(* PLC project PinDiagnosis, Hydac System GmbH PdtCodeBuilder.dll 1.2.7.80 *)
(* stored: companyURL http://www.hydac.com/, contentDescription This content was automatically generated. Please do not edit., creationDateTime 2025-04-18T16:40:50.760, version 1.0.0 *)

VAR_GLOBAL CONSTANT  (* Pins *)
  gc_PinList_C0 : ARRAY[0..95] OF POINTER TO TControllerPinProperties := [ADR(gc_Pin_C0_1), ADR(gc_Pin_C0_2), ADR(gc_Pin_C0_3), ADR(gc_Pin_C0_4), ADR(gc_Pin_C0_5), ADR(gc_Pin_C0_6), ADR(gc_Pin_C0_7), ADR(gc_Pin_C0_8), ADR(gc_Pin_C0_9), ADR(gc_Pin_C0_10), ADR(gc_Pin_C0_11), ADR(gc_Pin_C0_12), ADR(gc_Pin_C0_13), ADR(gc_Pin_C0_14), ADR(gc_Pin_C0_15), ADR(gc_Pin_C0_16), ADR(gc_Pin_C0_17), ADR(gc_Pin_C0_18), ADR(gc_Pin_C0_19), ADR(gc_Pin_C0_20), ADR(gc_Pin_C0_21), ADR(gc_Pin_C0_22), ADR(gc_Pin_C0_23), ADR(gc_Pin_C0_24), ADR(gc_Pin_C0_25), ADR(gc_Pin_C0_26), ADR(gc_Pin_C0_27), ADR(gc_Pin_C0_28), ADR(gc_Pin_C0_29), ADR(gc_Pin_C0_30), ADR(gc_Pin_C0_31), ADR(gc_Pin_C0_32), ADR(gc_Pin_C0_33), ADR(gc_Pin_C0_34), ADR(gc_Pin_C0_35), ADR(gc_Pin_C0_36), ADR(gc_Pin_C0_37), ADR(gc_Pin_C0_38), ADR(gc_Pin_C0_39), ADR(gc_Pin_C0_40), ADR(gc_Pin_C0_41), ADR(gc_Pin_C0_42), ADR(gc_Pin_C0_43), ADR(gc_Pin_C0_44), ADR(gc_Pin_C0_45), ADR(gc_Pin_C0_46), ADR(gc_Pin_C0_47), ADR(gc_Pin_C0_48), ADR(gc_Pin_C0_49), ADR(gc_Pin_C0_50), ADR(gc_Pin_C0_51), ADR(gc_Pin_C0_52), ADR(gc_Pin_C0_53), ADR(gc_Pin_C0_54), ADR(gc_Pin_C0_55), ADR(gc_Pin_C0_56), ADR(gc_Pin_C0_57), ADR(gc_Pin_C0_58), ADR(gc_Pin_C0_59), ADR(gc_Pin_C0_60), ADR(gc_Pin_C0_61), ADR(gc_Pin_C0_62), ADR(gc_Pin_C0_63), ADR(gc_Pin_C0_64), ADR(gc_Pin_C0_65), ADR(gc_Pin_C0_66), ADR(gc_Pin_C0_67), ADR(gc_Pin_C0_68), ADR(gc_Pin_C0_69), ADR(gc_Pin_C0_70), ADR(gc_Pin_C0_71), ADR(gc_Pin_C0_72), ADR(gc_Pin_C0_73), ADR(gc_Pin_C0_74), ADR(gc_Pin_C0_75), ADR(gc_Pin_C0_76), ADR(gc_Pin_C0_77), ADR(gc_Pin_C0_78), ADR(gc_Pin_C0_79), ADR(gc_Pin_C0_80), ADR(gc_Pin_C0_81), ADR(gc_Pin_C0_82), ADR(gc_Pin_C0_83), ADR(gc_Pin_C0_84), ADR(gc_Pin_C0_85), ADR(gc_Pin_C0_86), ADR(gc_Pin_C0_87), ADR(gc_Pin_C0_88), ADR(gc_Pin_C0_89), ADR(gc_Pin_C0_90), ADR(gc_Pin_C0_91), ADR(gc_Pin_C0_92), ADR(gc_Pin_C0_93), ADR(gc_Pin_C0_94), ADR(gc_Pin_C0_95), ADR(gc_Pin_C0_96)];
  gc_ControllerPinConfig_C0 : TControllerPinConfig := (EcuSA := 16#20, EcuName := 'C0', PinCount := 96, Pins := ADR(gc_PinList_C0));
  gc_PinList_C1 : ARRAY[0..95] OF POINTER TO TControllerPinProperties := [ADR(gc_Pin_C1_1), ADR(gc_Pin_C1_2), ADR(gc_Pin_C1_3), ADR(gc_Pin_C1_4), ADR(gc_Pin_C1_5), ADR(gc_Pin_C1_6), ADR(gc_Pin_C1_7), ADR(gc_Pin_C1_8), ADR(gc_Pin_C1_9), ADR(gc_Pin_C1_10), ADR(gc_Pin_C1_11), ADR(gc_Pin_C1_12), ADR(gc_Pin_C1_13), ADR(gc_Pin_C1_14), ADR(gc_Pin_C1_15), ADR(gc_Pin_C1_16), ADR(gc_Pin_C1_17), ADR(gc_Pin_C1_18), ADR(gc_Pin_C1_19), ADR(gc_Pin_C1_20), ADR(gc_Pin_C1_21), ADR(gc_Pin_C1_22), ADR(gc_Pin_C1_23), ADR(gc_Pin_C1_24), ADR(gc_Pin_C1_25), ADR(gc_Pin_C1_26), ADR(gc_Pin_C1_27), ADR(gc_Pin_C1_28), ADR(gc_Pin_C1_29), ADR(gc_Pin_C1_30), ADR(gc_Pin_C1_31), ADR(gc_Pin_C1_32), ADR(gc_Pin_C1_33), ADR(gc_Pin_C1_34), ADR(gc_Pin_C1_35), ADR(gc_Pin_C1_36), ADR(gc_Pin_C1_37), ADR(gc_Pin_C1_38), ADR(gc_Pin_C1_39), ADR(gc_Pin_C1_40), ADR(gc_Pin_C1_41), ADR(gc_Pin_C1_42), ADR(gc_Pin_C1_43), ADR(gc_Pin_C1_44), ADR(gc_Pin_C1_45), ADR(gc_Pin_C1_46), ADR(gc_Pin_C1_47), ADR(gc_Pin_C1_48), ADR(gc_Pin_C1_49), ADR(gc_Pin_C1_50), ADR(gc_Pin_C1_51), ADR(gc_Pin_C1_52), ADR(gc_Pin_C1_53), ADR(gc_Pin_C1_54), ADR(gc_Pin_C1_55), ADR(gc_Pin_C1_56), ADR(gc_Pin_C1_57), ADR(gc_Pin_C1_58), ADR(gc_Pin_C1_59), ADR(gc_Pin_C1_60), ADR(gc_Pin_C1_61), ADR(gc_Pin_C1_62), ADR(gc_Pin_C1_63), ADR(gc_Pin_C1_64), ADR(gc_Pin_C1_65), ADR(gc_Pin_C1_66), ADR(gc_Pin_C1_67), ADR(gc_Pin_C1_68), ADR(gc_Pin_C1_69), ADR(gc_Pin_C1_70), ADR(gc_Pin_C1_71), ADR(gc_Pin_C1_72), ADR(gc_Pin_C1_73), ADR(gc_Pin_C1_74), ADR(gc_Pin_C1_75), ADR(gc_Pin_C1_76), ADR(gc_Pin_C1_77), ADR(gc_Pin_C1_78), ADR(gc_Pin_C1_79), ADR(gc_Pin_C1_80), ADR(gc_Pin_C1_81), ADR(gc_Pin_C1_82), ADR(gc_Pin_C1_83), ADR(gc_Pin_C1_84), ADR(gc_Pin_C1_85), ADR(gc_Pin_C1_86), ADR(gc_Pin_C1_87), ADR(gc_Pin_C1_88), ADR(gc_Pin_C1_89), ADR(gc_Pin_C1_90), ADR(gc_Pin_C1_91), ADR(gc_Pin_C1_92), ADR(gc_Pin_C1_93), ADR(gc_Pin_C1_94), ADR(gc_Pin_C1_95), ADR(gc_Pin_C1_96)];
  gc_ControllerPinConfig_C1 : TControllerPinConfig := (EcuSA := 16#21, EcuName := 'C1', PinCount := 96, Pins := ADR(gc_PinList_C1));
  gc_ControllerPinConfigs : ARRAY[0..1] OF POINTER TO TControllerPinConfig := [ADR(gc_ControllerPinConfig_C0), ADR(gc_ControllerPinConfig_C1)];
END_VAR

VAR_GLOBAL CONSTANT  (* Pins_C0 *)
  gc_Pin_C0_1 : TControllerPinProperties := (Index := 1, Type_ := eControllerPinType.CIN, Number := '103', Mapping := eControllerPinMappingType.FIX, Symbol := '103', Info := 'Pressure Block Oscillaton Sensor', Description := 0);
  gc_Pin_C0_2 : TControllerPinProperties := (Index := 2, Type_ := eControllerPinType.CIN, Number := '104', Mapping := eControllerPinMappingType.FIX, Symbol := '104', Info := 'Temperature Transmission Sensor', Description := 0);
  gc_Pin_C0_3 : TControllerPinProperties := (Index := 3, Type_ := eControllerPinType.VIN, Number := '105', Mapping := eControllerPinMappingType.FIX, Symbol := '105', Info := 'Aru Radio 2 Contact', Description := 0);
  gc_Pin_C0_4 : TControllerPinProperties := (Index := 4, Type_ := eControllerPinType.VIN, Number := '106', Mapping := eControllerPinMappingType.FIX, Symbol := '106', Info := 'Vanne mat position basse NO', Description := 0);
  gc_Pin_C0_5 : TControllerPinProperties := (Index := 5, Type_ := eControllerPinType.CIN, Number := '127', Mapping := eControllerPinMappingType.FIX, Symbol := '127', Info := 'Pressure Brake Sensor', Description := 0);
  gc_Pin_C0_6 : TControllerPinProperties := (Index := 6, Type_ := eControllerPinType.VIN, Number := '128', Mapping := eControllerPinMappingType.FIX, Symbol := '128', Info := 'Aru Radio 1 Contact', Description := 0);
  gc_Pin_C0_7 : TControllerPinProperties := (Index := 7, Type_ := eControllerPinType.CIN, Number := '129', Mapping := eControllerPinMappingType.FIX, Symbol := '129', Info := 'Electric Pump Pressure', Description := 0);
  gc_Pin_C0_8 : TControllerPinProperties := (Index := 8, Type_ := eControllerPinType.VIN, Number := '130', Mapping := eControllerPinMappingType.FIX, Symbol := '130', Info := 'Capteur mat de position haute NC', Description := 0);
  gc_Pin_C0_9 : TControllerPinProperties := (Index := 9, Type_ := eControllerPinType.VIN, Number := '107', Mapping := eControllerPinMappingType.FIX, Symbol := '107', Info := 'Frame Rotation Sensor1', Description := 0);
  gc_Pin_C0_10 : TControllerPinProperties := (Index := 10, Type_ := eControllerPinType.VIN, Number := '131', Mapping := eControllerPinMappingType.FIX, Symbol := '131', Info := 'Down Oscillant Axle', Description := 0);
  gc_Pin_C0_11 : TControllerPinProperties := (Index := 11, Type_ := eControllerPinType.VIN, Number := '108', Mapping := eControllerPinMappingType.FIX, Symbol := '108', Info := 'Down Fixe Axle', Description := 0);
  gc_Pin_C0_12 : TControllerPinProperties := (Index := 12, Type_ := eControllerPinType.VIN, Number := '132', Mapping := eControllerPinMappingType.FIX, Symbol := '132', Info := 'Up Oscillant Axle', Description := 0);
  gc_Pin_C0_13 : TControllerPinProperties := (Index := 13, Type_ := eControllerPinType.VIN, Number := '109', Mapping := eControllerPinMappingType.FIX, Symbol := '109', Info := 'Up Fixe Axle', Description := 0);
  gc_Pin_C0_14 : TControllerPinProperties := (Index := 14, Type_ := eControllerPinType.VIN, Number := '133', Mapping := eControllerPinMappingType.FIX, Symbol := '133', Info := 'Frame Rotation Sensor 1', Description := 0);
  gc_Pin_C0_15 : TControllerPinProperties := (Index := 15, Type_ := eControllerPinType.VIN, Number := '110', Mapping := eControllerPinMappingType.FIX, Symbol := '110', Info := 'Rail Hook Sensor', Description := 0);
  gc_Pin_C0_16 : TControllerPinProperties := (Index := 16, Type_ := eControllerPinType.VIN, Number := '134', Mapping := eControllerPinMappingType.FIX, Symbol := '134', Info := 'Inductive Rail Sensor', Description := 0);
  gc_Pin_C0_17 : TControllerPinProperties := (Index := 17, Type_ := eControllerPinType.VIN, Number := '111', Mapping := eControllerPinMappingType.FIX, Symbol := '111', Info := 'Centered Turret', Description := 0);
  gc_Pin_C0_18 : TControllerPinProperties := (Index := 18, Type_ := eControllerPinType.VIN, Number := '135', Mapping := eControllerPinMappingType.FIX, Symbol := '135', Info := 'Work Key Track Side', Description := 0);
  gc_Pin_C0_19 : TControllerPinProperties := (Index := 19, Type_ := eControllerPinType.VIN, Number := '112', Mapping := eControllerPinMappingType.FIX, Symbol := '112', Info := 'Frame Rotation Sensor 2', Description := 0);
  gc_Pin_C0_20 : TControllerPinProperties := (Index := 20, Type_ := eControllerPinType.VIN, Number := '136', Mapping := eControllerPinMappingType.FIX, Symbol := '136', Info := 'Work Key Bilateral', Description := 0);
  gc_Pin_C0_21 : TControllerPinProperties := (Index := 21, Type_ := eControllerPinType.VIN, Number := '113', Mapping := eControllerPinMappingType.FIX, Symbol := '113', Info := 'Work Key Centered', Description := 0);
  gc_Pin_C0_22 : TControllerPinProperties := (Index := 22, Type_ := eControllerPinType.VIN, Number := '137', Mapping := eControllerPinMappingType.FIX, Symbol := '137', Info := 'Abutment Turret Track Side', Description := 0);
  gc_Pin_C0_23 : TControllerPinProperties := (Index := 23, Type_ := eControllerPinType.VIN, Number := '114', Mapping := eControllerPinMappingType.FIX, Symbol := '114', Info := 'Frame Rotation Sensor 2', Description := 0);
  gc_Pin_C0_24 : TControllerPinProperties := (Index := 24, Type_ := eControllerPinType.VIN, Number := '138', Mapping := eControllerPinMappingType.FIX, Symbol := '138', Info := 'Abutment Turret Centred Side', Description := 0);
  gc_Pin_C0_25 : TControllerPinProperties := (Index := 25, Type_ := eControllerPinType.CPX, Number := '115', Mapping := eControllerPinMappingType.BLO, Symbol := '115', Info := 'Oscillant Axle Speed Sensor', Description := 0);
  gc_Pin_C0_26 : TControllerPinProperties := (Index := 26, Type_ := eControllerPinType.VIN, Number := '139', Mapping := eControllerPinMappingType.FIX, Symbol := '139', Info := 'Oscillant Axle Speed Sensor Dir', Description := 0);
  gc_Pin_C0_27 : TControllerPinProperties := (Index := 27, Type_ := eControllerPinType.CPX, Number := '116', Mapping := eControllerPinMappingType.BLO, Symbol := '116', Info := 'Fixe Axle Speed Sensor', Description := 0);
  gc_Pin_C0_28 : TControllerPinProperties := (Index := 28, Type_ := eControllerPinType.VIN, Number := '140', Mapping := eControllerPinMappingType.FIX, Symbol := '140', Info := 'Fixe Axle Speed Sensor Dir', Description := 0);
  gc_Pin_C0_29 : TControllerPinProperties := (Index := 29, Type_ := eControllerPinType.VIN, Number := '117', Mapping := eControllerPinMappingType.FIX, Symbol := '117', Info := 'Trailer Gache', Description := 0);
  gc_Pin_C0_30 : TControllerPinProperties := (Index := 30, Type_ := eControllerPinType.VIN, Number := '141', Mapping := eControllerPinMappingType.FIX, Symbol := '141', Info := 'Measuring Mast Sensor Folded', Description := 0);
  gc_Pin_C0_31 : TControllerPinProperties := (Index := 31, Type_ := eControllerPinType.VIN, Number := '122', Mapping := eControllerPinMappingType.FIX, Symbol := '122', Info := 'PIN_122', Description := 0);
  gc_Pin_C0_32 : TControllerPinProperties := (Index := 32, Type_ := eControllerPinType.VIN, Number := '146', Mapping := eControllerPinMappingType.FIX, Symbol := '146', Info := 'PIN_146', Description := 0);
  gc_Pin_C0_33 : TControllerPinProperties := (Index := 33, Type_ := eControllerPinType.VIN, Number := '123', Mapping := eControllerPinMappingType.FIX, Symbol := '123', Info := 'PIN_123', Description := 0);
  gc_Pin_C0_34 : TControllerPinProperties := (Index := 34, Type_ := eControllerPinType.VIN, Number := '147', Mapping := eControllerPinMappingType.FIX, Symbol := '147', Info := 'PIN_147', Description := 0);
  gc_Pin_C0_35 : TControllerPinProperties := (Index := 35, Type_ := eControllerPinType.VIN, Number := '124', Mapping := eControllerPinMappingType.FIX, Symbol := '124', Info := 'Aru 1 Contact', Description := 0);
  gc_Pin_C0_36 : TControllerPinProperties := (Index := 36, Type_ := eControllerPinType.VIN, Number := '148', Mapping := eControllerPinMappingType.FIX, Symbol := '148', Info := 'Aru 2 Contact', Description := 0);
  gc_Pin_C0_37 : TControllerPinProperties := (Index := 37, Type_ := eControllerPinType.DOU, Number := '153', Mapping := eControllerPinMappingType.FIX, Symbol := '153', Info := 'Ev Deflector Transmission', Description := 0);
  gc_Pin_C0_38 : TControllerPinProperties := (Index := 38, Type_ := eControllerPinType.DOU, Number := '177', Mapping := eControllerPinMappingType.FIX, Symbol := '177', Info := 'Ev Unblock OScillation Axle', Description := 0);
  gc_Pin_C0_39 : TControllerPinProperties := (Index := 39, Type_ := eControllerPinType.DOU, Number := '156', Mapping := eControllerPinMappingType.FIX, Symbol := '156', Info := 'SupplyAnaSensors', Description := 0);
  gc_Pin_C0_40 : TControllerPinProperties := (Index := 40, Type_ := eControllerPinType.NA, Number := '180', Mapping := eControllerPinMappingType.CHA, Symbol := '180', Info := 'PIN_180', Description := 0);
  gc_Pin_C0_41 : TControllerPinProperties := (Index := 41, Type_ := eControllerPinType.DOU, Number := '159', Mapping := eControllerPinMappingType.FIX, Symbol := '159', Info := 'Ev2 Deflector Transmission', Description := 0);
  gc_Pin_C0_42 : TControllerPinProperties := (Index := 42, Type_ := eControllerPinType.NA, Number := '183', Mapping := eControllerPinMappingType.CHA, Symbol := '183', Info := 'PIN_183', Description := 0);
  gc_Pin_C0_43 : TControllerPinProperties := (Index := 43, Type_ := eControllerPinType.DOU, Number := '186', Mapping := eControllerPinMappingType.FIX, Symbol := '186', Info := 'Ev Park Brake Axle Oscillant', Description := 0);
  gc_Pin_C0_44 : TControllerPinProperties := (Index := 44, Type_ := eControllerPinType.DOU, Number := '162', Mapping := eControllerPinMappingType.FIX, Symbol := '162', Info := 'Ev Park Brake Axle Fixe', Description := 0);
  gc_Pin_C0_45 : TControllerPinProperties := (Index := 45, Type_ := eControllerPinType.DOU, Number := '189', Mapping := eControllerPinMappingType.FIX, Symbol := '189', Info := 'Ev Service Brake Axle OScillant', Description := 0);
  gc_Pin_C0_46 : TControllerPinProperties := (Index := 46, Type_ := eControllerPinType.DOU, Number := '165', Mapping := eControllerPinMappingType.FIX, Symbol := '165', Info := 'Ev Service Brake Axle Fixe', Description := 0);
  gc_Pin_C0_47 : TControllerPinProperties := (Index := 47, Type_ := eControllerPinType.DOU, Number := '192', Mapping := eControllerPinMappingType.FIX, Symbol := '192', Info := 'Ev 2nd Park Brake Axle Fixe', Description := 0);
  gc_Pin_C0_48 : TControllerPinProperties := (Index := 48, Type_ := eControllerPinType.DOU, Number := '168', Mapping := eControllerPinMappingType.FIX, Symbol := '168', Info := 'Ev 2nd Park Brake Axle Osci', Description := 0);
  gc_Pin_C0_49 : TControllerPinProperties := (Index := 49, Type_ := eControllerPinType.DOU, Number := '195', Mapping := eControllerPinMappingType.FIX, Symbol := '195', Info := 'Ev Service Brake Track', Description := 0);
  gc_Pin_C0_50 : TControllerPinProperties := (Index := 50, Type_ := eControllerPinType.DOU, Number := '171', Mapping := eControllerPinMappingType.FIX, Symbol := '171', Info := 'Ev Power Reduction', Description := 0);
  gc_Pin_C0_51 : TControllerPinProperties := (Index := 51, Type_ := eControllerPinType.DOU, Number := '154', Mapping := eControllerPinMappingType.FIX, Symbol := '154', Info := 'Neon Lights', Description := 0);
  gc_Pin_C0_52 : TControllerPinProperties := (Index := 52, Type_ := eControllerPinType.NA, Number := '178', Mapping := eControllerPinMappingType.CHA, Symbol := '178', Info := 'PIN_178', Description := 0);
  gc_Pin_C0_53 : TControllerPinProperties := (Index := 53, Type_ := eControllerPinType.NA, Number := '157', Mapping := eControllerPinMappingType.CHA, Symbol := '157', Info := 'PIN_157', Description := 0);
  gc_Pin_C0_54 : TControllerPinProperties := (Index := 54, Type_ := eControllerPinType.NA, Number := '181', Mapping := eControllerPinMappingType.CHA, Symbol := '181', Info := 'PIN_181', Description := 0);
  gc_Pin_C0_55 : TControllerPinProperties := (Index := 55, Type_ := eControllerPinType.DOU, Number := '160', Mapping := eControllerPinMappingType.FIX, Symbol := '160', Info := 'Supply Radio Receiver', Description := 0);
  gc_Pin_C0_56 : TControllerPinProperties := (Index := 56, Type_ := eControllerPinType.DOU, Number := '184', Mapping := eControllerPinMappingType.FIX, Symbol := '184', Info := 'Buzzer Lynx Moving Machine', Description := 0);
  gc_Pin_C0_57 : TControllerPinProperties := (Index := 57, Type_ := eControllerPinType.DOU, Number := '187', Mapping := eControllerPinMappingType.FIX, Symbol := '187', Info := 'Ev Dev Rail electric mode', Description := 0);
  gc_Pin_C0_58 : TControllerPinProperties := (Index := 58, Type_ := eControllerPinType.DOU, Number := '163', Mapping := eControllerPinMappingType.FIX, Symbol := '163', Info := 'Klaxon Neotec', Description := 0);
  gc_Pin_C0_59 : TControllerPinProperties := (Index := 59, Type_ := eControllerPinType.DOU, Number := '190', Mapping := eControllerPinMappingType.FIX, Symbol := '190', Info := 'Ev Up Measuring Mast', Description := 0);
  gc_Pin_C0_60 : TControllerPinProperties := (Index := 60, Type_ := eControllerPinType.DOU, Number := '166', Mapping := eControllerPinMappingType.FIX, Symbol := '166', Info := 'Ev Down Measuring Mast', Description := 0);
  gc_Pin_C0_61 : TControllerPinProperties := (Index := 61, Type_ := eControllerPinType.DOU, Number := '193', Mapping := eControllerPinMappingType.FIX, Symbol := '193', Info := 'Ev Up Axle Oscillant', Description := 0);
  gc_Pin_C0_62 : TControllerPinProperties := (Index := 62, Type_ := eControllerPinType.DOU, Number := '169', Mapping := eControllerPinMappingType.FIX, Symbol := '169', Info := 'Ev Down Axle Oscillant', Description := 0);
  gc_Pin_C0_63 : TControllerPinProperties := (Index := 63, Type_ := eControllerPinType.DOU, Number := '196', Mapping := eControllerPinMappingType.FIX, Symbol := '196', Info := 'Ev Up Axle Fixe', Description := 0);
  gc_Pin_C0_64 : TControllerPinProperties := (Index := 64, Type_ := eControllerPinType.DOU, Number := '172', Mapping := eControllerPinMappingType.FIX, Symbol := '172', Info := 'Ev Down Axle Fixe', Description := 0);
  gc_Pin_C0_65 : TControllerPinProperties := (Index := 65, Type_ := eControllerPinType.PWM, Number := '101', Mapping := eControllerPinMappingType.FIX, Symbol := '101', Info := 'Ev Forward Pump', Description := 0);
  gc_Pin_C0_66 : TControllerPinProperties := (Index := 66, Type_ := eControllerPinType.PWM, Number := '125', Mapping := eControllerPinMappingType.FIX, Symbol := '125', Info := 'Ev Backward Pump', Description := 0);
  gc_Pin_C0_67 : TControllerPinProperties := (Index := 67, Type_ := eControllerPinType.DOU, Number := '150', Mapping := eControllerPinMappingType.FIX, Symbol := '150', Info := 'PIN_150', Description := 0);
  gc_Pin_C0_68 : TControllerPinProperties := (Index := 68, Type_ := eControllerPinType.NA, Number := '174', Mapping := eControllerPinMappingType.CHA, Symbol := '174', Info := 'PIN_174', Description := 0);
  gc_Pin_C0_69 : TControllerPinProperties := (Index := 69, Type_ := eControllerPinType.NA, Number := '102', Mapping := eControllerPinMappingType.CHA, Symbol := '102', Info := 'PIN_102', Description := 0);
  gc_Pin_C0_70 : TControllerPinProperties := (Index := 70, Type_ := eControllerPinType.DOU, Number := '126', Mapping := eControllerPinMappingType.FIX, Symbol := '126', Info := 'PIN_126', Description := 0);
  gc_Pin_C0_71 : TControllerPinProperties := (Index := 71, Type_ := eControllerPinType.NA, Number := '151', Mapping := eControllerPinMappingType.CHA, Symbol := '151', Info := 'PIN_151', Description := 0);
  gc_Pin_C0_72 : TControllerPinProperties := (Index := 72, Type_ := eControllerPinType.DOU, Number := '175', Mapping := eControllerPinMappingType.FIX, Symbol := '175', Info := 'PIN_175', Description := 0);
  gc_Pin_C0_73 : TControllerPinProperties := (Index := 73, Type_ := eControllerPinType.DOU, Number := '149', Mapping := eControllerPinMappingType.FIX, Symbol := '149', Info := 'White Light AVG', Description := 0);
  gc_Pin_C0_74 : TControllerPinProperties := (Index := 74, Type_ := eControllerPinType.DOU, Number := '173', Mapping := eControllerPinMappingType.FIX, Symbol := '173', Info := 'White Light AVD', Description := 0);
  gc_Pin_C0_75 : TControllerPinProperties := (Index := 75, Type_ := eControllerPinType.DOU, Number := '152', Mapping := eControllerPinMappingType.FIX, Symbol := '152', Info := 'Red Light AVG', Description := 0);
  gc_Pin_C0_76 : TControllerPinProperties := (Index := 76, Type_ := eControllerPinType.DOU, Number := '176', Mapping := eControllerPinMappingType.FIX, Symbol := '176', Info := 'Red Light AVD', Description := 0);
  gc_Pin_C0_77 : TControllerPinProperties := (Index := 77, Type_ := eControllerPinType.DOU, Number := '155', Mapping := eControllerPinMappingType.FIX, Symbol := '155', Info := 'White Light ARG', Description := 0);
  gc_Pin_C0_78 : TControllerPinProperties := (Index := 78, Type_ := eControllerPinType.DOU, Number := '179', Mapping := eControllerPinMappingType.FIX, Symbol := '179', Info := 'White Light ARD', Description := 0);
  gc_Pin_C0_79 : TControllerPinProperties := (Index := 79, Type_ := eControllerPinType.DOU, Number := '158', Mapping := eControllerPinMappingType.FIX, Symbol := '158', Info := 'Red Light ARG', Description := 0);
  gc_Pin_C0_80 : TControllerPinProperties := (Index := 80, Type_ := eControllerPinType.DOU, Number := '182', Mapping := eControllerPinMappingType.FIX, Symbol := '182', Info := 'Red Light ARD', Description := 0);
  gc_Pin_C0_81 : TControllerPinProperties := (Index := 81, Type_ := eControllerPinType.DOU, Number := '251', Mapping := eControllerPinMappingType.FIX, Symbol := '251', Info := 'Return low side Ev Forward Pump', Description := 0);
  gc_Pin_C0_82 : TControllerPinProperties := (Index := 82, Type_ := eControllerPinType.DOU, Number := '238', Mapping := eControllerPinMappingType.FIX, Symbol := '238', Info := 'Return low side Ev Backward Pump', Description := 0);
  gc_Pin_C0_83 : TControllerPinProperties := (Index := 83, Type_ := eControllerPinType.DOU, Number := '252', Mapping := eControllerPinMappingType.FIX, Symbol := '252', Info := 'Pvg Left Track Lowside', Description := 0);
  gc_Pin_C0_84 : TControllerPinProperties := (Index := 84, Type_ := eControllerPinType.DOU, Number := '239', Mapping := eControllerPinMappingType.FIX, Symbol := '239', Info := 'PVg Right Track Lowside', Description := 0);
  gc_Pin_C0_85 : TControllerPinProperties := (Index := 85, Type_ := eControllerPinType.NA, Number := '253', Mapping := eControllerPinMappingType.CHA, Symbol := '253', Info := 'PIN_253', Description := 0);
  gc_Pin_C0_86 : TControllerPinProperties := (Index := 86, Type_ := eControllerPinType.NA, Number := '240', Mapping := eControllerPinMappingType.CHA, Symbol := '240', Info := 'PIN_240', Description := 0);
  gc_Pin_C0_87 : TControllerPinProperties := (Index := 87, Type_ := eControllerPinType.NA, Number := '254', Mapping := eControllerPinMappingType.CHA, Symbol := '254', Info := 'PIN_254', Description := 0);
  gc_Pin_C0_88 : TControllerPinProperties := (Index := 88, Type_ := eControllerPinType.NA, Number := '241', Mapping := eControllerPinMappingType.CHA, Symbol := '241', Info := 'PIN_241', Description := 0);
  gc_Pin_C0_89 : TControllerPinProperties := (Index := 89, Type_ := eControllerPinType.VOU, Number := '161', Mapping := eControllerPinMappingType.FIX, Symbol := '161', Info := 'Pvg Left Track', Description := 0);
  gc_Pin_C0_90 : TControllerPinProperties := (Index := 90, Type_ := eControllerPinType.VOU, Number := '185', Mapping := eControllerPinMappingType.FIX, Symbol := '185', Info := 'Pvg Right Track', Description := 0);
  gc_Pin_C0_91 : TControllerPinProperties := (Index := 91, Type_ := eControllerPinType.DOU, Number := '188', Mapping := eControllerPinMappingType.FIX, Symbol := '188', Info := 'Supply Pvg Left Track', Description := 0);
  gc_Pin_C0_92 : TControllerPinProperties := (Index := 92, Type_ := eControllerPinType.DOU, Number := '164', Mapping := eControllerPinMappingType.FIX, Symbol := '164', Info := 'Supply Pvg Right Track', Description := 0);
  gc_Pin_C0_93 : TControllerPinProperties := (Index := 93, Type_ := eControllerPinType.VOU, Number := '191', Mapping := eControllerPinMappingType.FIX, Symbol := '191', Info := 'Pvg Trans Rail Electric', Description := 0);
  gc_Pin_C0_94 : TControllerPinProperties := (Index := 94, Type_ := eControllerPinType.DOU, Number := '167', Mapping := eControllerPinMappingType.FIX, Symbol := '167', Info := 'Supply Pvg Trans Rail Electric', Description := 0);
  gc_Pin_C0_95 : TControllerPinProperties := (Index := 95, Type_ := eControllerPinType.DOU, Number := '194', Mapping := eControllerPinMappingType.FIX, Symbol := '194', Info := 'White Trailer Lights', Description := 0);
  gc_Pin_C0_96 : TControllerPinProperties := (Index := 96, Type_ := eControllerPinType.DOU, Number := '170', Mapping := eControllerPinMappingType.FIX, Symbol := '170', Info := 'Red Trailer Lights', Description := 0);
END_VAR

VAR_GLOBAL CONSTANT  (* Pins_C1 *)
  gc_Pin_C1_1 : TControllerPinProperties := (Index := 1, Type_ := eControllerPinType.CIN, Number := '103', Mapping := eControllerPinMappingType.FIX, Symbol := '103', Info := 'Transmission 1 pressure sensor', Description := 0);
  gc_Pin_C1_2 : TControllerPinProperties := (Index := 2, Type_ := eControllerPinType.CIN, Number := '104', Mapping := eControllerPinMappingType.FIX, Symbol := '104', Info := 'Delta arm 1 angular sensor', Description := 0);
  gc_Pin_C1_3 : TControllerPinProperties := (Index := 3, Type_ := eControllerPinType.CIN, Number := '105', Mapping := eControllerPinMappingType.FIX, Symbol := '105', Info := 'Arrow arm 1 angular sensor', Description := 0);
  gc_Pin_C1_4 : TControllerPinProperties := (Index := 4, Type_ := eControllerPinType.RES, Number := '106', Mapping := eControllerPinMappingType.FIX, Symbol := '106', Info := 'Gas gauge', Description := 0);
  gc_Pin_C1_5 : TControllerPinProperties := (Index := 5, Type_ := eControllerPinType.CIN, Number := '127', Mapping := eControllerPinMappingType.FIX, Symbol := '127', Info := 'Transmission 2 pressure sensor', Description := 0);
  gc_Pin_C1_6 : TControllerPinProperties := (Index := 6, Type_ := eControllerPinType.CIN, Number := '128', Mapping := eControllerPinMappingType.FIX, Symbol := '128', Info := 'Delta arm 2 angular sensor', Description := 0);
  gc_Pin_C1_7 : TControllerPinProperties := (Index := 7, Type_ := eControllerPinType.CIN, Number := '129', Mapping := eControllerPinMappingType.FIX, Symbol := '129', Info := 'Arrow arm 2 angular sensor', Description := 0);
  gc_Pin_C1_8 : TControllerPinProperties := (Index := 8, Type_ := eControllerPinType.CIN, Number := '130', Mapping := eControllerPinMappingType.FIX, Symbol := '130', Info := 'Bypass Pressure Sensor', Description := 0);
  gc_Pin_C1_9 : TControllerPinProperties := (Index := 9, Type_ := eControllerPinType.NA, Number := '107', Mapping := eControllerPinMappingType.CHA, Symbol := '107', Info := 'PIN_107', Description := 0);
  gc_Pin_C1_10 : TControllerPinProperties := (Index := 10, Type_ := eControllerPinType.VIN, Number := '131', Mapping := eControllerPinMappingType.FIX, Symbol := '131', Info := 'Turret post selector', Description := 0);
  gc_Pin_C1_11 : TControllerPinProperties := (Index := 11, Type_ := eControllerPinType.VIN, Number := '108', Mapping := eControllerPinMappingType.FIX, Symbol := '108', Info := 'Radio post selector', Description := 0);
  gc_Pin_C1_12 : TControllerPinProperties := (Index := 12, Type_ := eControllerPinType.VIN, Number := '132', Mapping := eControllerPinMappingType.FIX, Symbol := '132', Info := 'Nacelle post selector', Description := 0);
  gc_Pin_C1_13 : TControllerPinProperties := (Index := 13, Type_ := eControllerPinType.NA, Number := '109', Mapping := eControllerPinMappingType.CHA, Symbol := '109', Info := 'PIN_109', Description := 0);
  gc_Pin_C1_14 : TControllerPinProperties := (Index := 14, Type_ := eControllerPinType.NA, Number := '133', Mapping := eControllerPinMappingType.CHA, Symbol := '133', Info := 'PIN_133', Description := 0);
  gc_Pin_C1_15 : TControllerPinProperties := (Index := 15, Type_ := eControllerPinType.CIN, Number := '110', Mapping := eControllerPinMappingType.FIX, Symbol := '110', Info := 'Temperature  reservoir d huile', Description := 0);
  gc_Pin_C1_16 : TControllerPinProperties := (Index := 16, Type_ := eControllerPinType.NA, Number := '134', Mapping := eControllerPinMappingType.CHA, Symbol := '134', Info := 'PIN_134', Description := 0);
  gc_Pin_C1_17 : TControllerPinProperties := (Index := 17, Type_ := eControllerPinType.VIN, Number := '111', Mapping := eControllerPinMappingType.FIX, Symbol := '111', Info := 'Fault pvg delta arm', Description := 0);
  gc_Pin_C1_18 : TControllerPinProperties := (Index := 18, Type_ := eControllerPinType.VIN, Number := '135', Mapping := eControllerPinMappingType.FIX, Symbol := '135', Info := 'Fault pvg boom arm', Description := 0);
  gc_Pin_C1_19 : TControllerPinProperties := (Index := 19, Type_ := eControllerPinType.VIN, Number := '112', Mapping := eControllerPinMappingType.FIX, Symbol := '112', Info := 'Fault pvg telescope arm', Description := 0);
  gc_Pin_C1_20 : TControllerPinProperties := (Index := 20, Type_ := eControllerPinType.VIN, Number := '136', Mapping := eControllerPinMappingType.FIX, Symbol := '136', Info := 'Fault pvg ev pro tor', Description := 0);
  gc_Pin_C1_21 : TControllerPinProperties := (Index := 21, Type_ := eControllerPinType.NA, Number := '113', Mapping := eControllerPinMappingType.CHA, Symbol := '113', Info := 'PIN_113', Description := 0);
  gc_Pin_C1_22 : TControllerPinProperties := (Index := 22, Type_ := eControllerPinType.VIN, Number := '137', Mapping := eControllerPinMappingType.FIX, Symbol := '137', Info := 'Aru1', Description := 0);
  gc_Pin_C1_23 : TControllerPinProperties := (Index := 23, Type_ := eControllerPinType.NA, Number := '114', Mapping := eControllerPinMappingType.CHA, Symbol := '114', Info := 'PIN_114', Description := 0);
  gc_Pin_C1_24 : TControllerPinProperties := (Index := 24, Type_ := eControllerPinType.VIN, Number := '138', Mapping := eControllerPinMappingType.FIX, Symbol := '138', Info := 'Aru2', Description := 0);
  gc_Pin_C1_25 : TControllerPinProperties := (Index := 25, Type_ := eControllerPinType.NA, Number := '115', Mapping := eControllerPinMappingType.CHA, Symbol := '115', Info := 'PIN_115', Description := 0);
  gc_Pin_C1_26 : TControllerPinProperties := (Index := 26, Type_ := eControllerPinType.NA, Number := '139', Mapping := eControllerPinMappingType.CHA, Symbol := '139', Info := 'PIN_139', Description := 0);
  gc_Pin_C1_27 : TControllerPinProperties := (Index := 27, Type_ := eControllerPinType.NA, Number := '116', Mapping := eControllerPinMappingType.CHA, Symbol := '116', Info := 'PIN_116', Description := 0);
  gc_Pin_C1_28 : TControllerPinProperties := (Index := 28, Type_ := eControllerPinType.NA, Number := '140', Mapping := eControllerPinMappingType.CHA, Symbol := '140', Info := 'PIN_140', Description := 0);
  gc_Pin_C1_29 : TControllerPinProperties := (Index := 29, Type_ := eControllerPinType.VIN, Number := '117', Mapping := eControllerPinMappingType.FIX, Symbol := '117', Info := 'Delta arm floded sensor', Description := 0);
  gc_Pin_C1_30 : TControllerPinProperties := (Index := 30, Type_ := eControllerPinType.VIN, Number := '141', Mapping := eControllerPinMappingType.FIX, Symbol := '141', Info := 'Boom arm folded sensor', Description := 0);
  gc_Pin_C1_31 : TControllerPinProperties := (Index := 31, Type_ := eControllerPinType.VIN, Number := '122', Mapping := eControllerPinMappingType.FIX, Symbol := '122', Info := 'Entry telescope Fdc Sensor', Description := 0);
  gc_Pin_C1_32 : TControllerPinProperties := (Index := 32, Type_ := eControllerPinType.NA, Number := '146', Mapping := eControllerPinMappingType.CHA, Symbol := '146', Info := 'PIN_146', Description := 0);
  gc_Pin_C1_33 : TControllerPinProperties := (Index := 33, Type_ := eControllerPinType.NA, Number := '123', Mapping := eControllerPinMappingType.CHA, Symbol := '123', Info := 'PIN_123', Description := 0);
  gc_Pin_C1_34 : TControllerPinProperties := (Index := 34, Type_ := eControllerPinType.VIN, Number := '147', Mapping := eControllerPinMappingType.FIX, Symbol := '147', Info := 'PIN_147', Description := 0);
  gc_Pin_C1_35 : TControllerPinProperties := (Index := 35, Type_ := eControllerPinType.VIN, Number := '124', Mapping := eControllerPinMappingType.FIX, Symbol := '124', Info := 'Active help', Description := 0);
  gc_Pin_C1_36 : TControllerPinProperties := (Index := 36, Type_ := eControllerPinType.VIN, Number := '148', Mapping := eControllerPinMappingType.FIX, Symbol := '148', Info := 'Alternator charge OK', Description := 0);
  gc_Pin_C1_37 : TControllerPinProperties := (Index := 37, Type_ := eControllerPinType.DOU, Number := '153', Mapping := eControllerPinMappingType.FIX, Symbol := '153', Info := 'Suplly Ana Sensors', Description := 0);
  gc_Pin_C1_38 : TControllerPinProperties := (Index := 38, Type_ := eControllerPinType.DOU, Number := '177', Mapping := eControllerPinMappingType.FIX, Symbol := '177', Info := 'PIN_177', Description := 0);
  gc_Pin_C1_39 : TControllerPinProperties := (Index := 39, Type_ := eControllerPinType.NA, Number := '156', Mapping := eControllerPinMappingType.CHA, Symbol := '156', Info := 'PIN_156', Description := 0);
  gc_Pin_C1_40 : TControllerPinProperties := (Index := 40, Type_ := eControllerPinType.PWM, Number := '180', Mapping := eControllerPinMappingType.FIX, Symbol := '180', Info := 'Ev prop generator', Description := 0);
  gc_Pin_C1_41 : TControllerPinProperties := (Index := 41, Type_ := eControllerPinType.DOU, Number := '159', Mapping := eControllerPinMappingType.FIX, Symbol := '159', Info := 'Ev sync rotation', Description := 0);
  gc_Pin_C1_42 : TControllerPinProperties := (Index := 42, Type_ := eControllerPinType.DOU, Number := '183', Mapping := eControllerPinMappingType.FIX, Symbol := '183', Info := 'Noisemarker', Description := 0);
  gc_Pin_C1_43 : TControllerPinProperties := (Index := 43, Type_ := eControllerPinType.DOU, Number := '186', Mapping := eControllerPinMappingType.FIX, Symbol := '186', Info := 'PIN_186', Description := 0);
  gc_Pin_C1_44 : TControllerPinProperties := (Index := 44, Type_ := eControllerPinType.DOU, Number := '162', Mapping := eControllerPinMappingType.FIX, Symbol := '162', Info := 'PIN_162', Description := 0);
  gc_Pin_C1_45 : TControllerPinProperties := (Index := 45, Type_ := eControllerPinType.NA, Number := '189', Mapping := eControllerPinMappingType.CHA, Symbol := '189', Info := 'PIN_189', Description := 0);
  gc_Pin_C1_46 : TControllerPinProperties := (Index := 46, Type_ := eControllerPinType.NA, Number := '165', Mapping := eControllerPinMappingType.CHA, Symbol := '165', Info := 'PIN_165', Description := 0);
  gc_Pin_C1_47 : TControllerPinProperties := (Index := 47, Type_ := eControllerPinType.NA, Number := '192', Mapping := eControllerPinMappingType.CHA, Symbol := '192', Info := 'PIN_192', Description := 0);
  gc_Pin_C1_48 : TControllerPinProperties := (Index := 48, Type_ := eControllerPinType.NA, Number := '168', Mapping := eControllerPinMappingType.CHA, Symbol := '168', Info := 'PIN_168', Description := 0);
  gc_Pin_C1_49 : TControllerPinProperties := (Index := 49, Type_ := eControllerPinType.NA, Number := '195', Mapping := eControllerPinMappingType.CHA, Symbol := '195', Info := 'PIN_195', Description := 0);
  gc_Pin_C1_50 : TControllerPinProperties := (Index := 50, Type_ := eControllerPinType.NA, Number := '171', Mapping := eControllerPinMappingType.CHA, Symbol := '171', Info := 'PIN_171', Description := 0);
  gc_Pin_C1_51 : TControllerPinProperties := (Index := 51, Type_ := eControllerPinType.DOU, Number := '154', Mapping := eControllerPinMappingType.FIX, Symbol := '154', Info := 'Ev rotation turret clockwise', Description := 0);
  gc_Pin_C1_52 : TControllerPinProperties := (Index := 52, Type_ := eControllerPinType.DOU, Number := '178', Mapping := eControllerPinMappingType.FIX, Symbol := '178', Info := 'Ev rotation turret counter clockwise', Description := 0);
  gc_Pin_C1_53 : TControllerPinProperties := (Index := 53, Type_ := eControllerPinType.DOU, Number := '157', Mapping := eControllerPinMappingType.FIX, Symbol := '157', Info := 'Ev roration basket counter clockwise', Description := 0);
  gc_Pin_C1_54 : TControllerPinProperties := (Index := 54, Type_ := eControllerPinType.DOU, Number := '181', Mapping := eControllerPinMappingType.FIX, Symbol := '181', Info := 'Ev rotation basket clokwise', Description := 0);
  gc_Pin_C1_55 : TControllerPinProperties := (Index := 55, Type_ := eControllerPinType.DOU, Number := '160', Mapping := eControllerPinMappingType.FIX, Symbol := '160', Info := 'Ev up pendular', Description := 0);
  gc_Pin_C1_56 : TControllerPinProperties := (Index := 56, Type_ := eControllerPinType.DOU, Number := '184', Mapping := eControllerPinMappingType.FIX, Symbol := '184', Info := 'Ev down pendular', Description := 0);
  gc_Pin_C1_57 : TControllerPinProperties := (Index := 57, Type_ := eControllerPinType.DOU, Number := '187', Mapping := eControllerPinMappingType.FIX, Symbol := '187', Info := 'Ev up inclinaison basket', Description := 0);
  gc_Pin_C1_58 : TControllerPinProperties := (Index := 58, Type_ := eControllerPinType.DOU, Number := '163', Mapping := eControllerPinMappingType.FIX, Symbol := '163', Info := 'Ev down inclinaison basket', Description := 0);
  gc_Pin_C1_59 : TControllerPinProperties := (Index := 59, Type_ := eControllerPinType.NA, Number := '190', Mapping := eControllerPinMappingType.CHA, Symbol := '190', Info := 'PIN_190', Description := 0);
  gc_Pin_C1_60 : TControllerPinProperties := (Index := 60, Type_ := eControllerPinType.NA, Number := '166', Mapping := eControllerPinMappingType.CHA, Symbol := '166', Info := 'PIN_166', Description := 0);
  gc_Pin_C1_61 : TControllerPinProperties := (Index := 61, Type_ := eControllerPinType.NA, Number := '193', Mapping := eControllerPinMappingType.CHA, Symbol := '193', Info := 'PIN_193', Description := 0);
  gc_Pin_C1_62 : TControllerPinProperties := (Index := 62, Type_ := eControllerPinType.NA, Number := '169', Mapping := eControllerPinMappingType.CHA, Symbol := '169', Info := 'PIN_169', Description := 0);
  gc_Pin_C1_63 : TControllerPinProperties := (Index := 63, Type_ := eControllerPinType.NA, Number := '196', Mapping := eControllerPinMappingType.CHA, Symbol := '196', Info := 'PIN_196', Description := 0);
  gc_Pin_C1_64 : TControllerPinProperties := (Index := 64, Type_ := eControllerPinType.NA, Number := '172', Mapping := eControllerPinMappingType.CHA, Symbol := '172', Info := 'PIN_172', Description := 0);
  gc_Pin_C1_65 : TControllerPinProperties := (Index := 65, Type_ := eControllerPinType.NA, Number := '101', Mapping := eControllerPinMappingType.CHA, Symbol := '101', Info := 'PIN_101', Description := 0);
  gc_Pin_C1_66 : TControllerPinProperties := (Index := 66, Type_ := eControllerPinType.NA, Number := '125', Mapping := eControllerPinMappingType.CHA, Symbol := '125', Info := 'PIN_125', Description := 0);
  gc_Pin_C1_67 : TControllerPinProperties := (Index := 67, Type_ := eControllerPinType.NA, Number := '150', Mapping := eControllerPinMappingType.CHA, Symbol := '150', Info := 'PIN_150', Description := 0);
  gc_Pin_C1_68 : TControllerPinProperties := (Index := 68, Type_ := eControllerPinType.NA, Number := '174', Mapping := eControllerPinMappingType.CHA, Symbol := '174', Info := 'Regime motor alternator', Description := 0);
  gc_Pin_C1_69 : TControllerPinProperties := (Index := 69, Type_ := eControllerPinType.NA, Number := '102', Mapping := eControllerPinMappingType.CHA, Symbol := '102', Info := 'PIN_102', Description := 0);
  gc_Pin_C1_70 : TControllerPinProperties := (Index := 70, Type_ := eControllerPinType.NA, Number := '126', Mapping := eControllerPinMappingType.CHA, Symbol := '126', Info := 'PIN_126', Description := 0);
  gc_Pin_C1_71 : TControllerPinProperties := (Index := 71, Type_ := eControllerPinType.NA, Number := '151', Mapping := eControllerPinMappingType.CHA, Symbol := '151', Info := 'PIN_151', Description := 0);
  gc_Pin_C1_72 : TControllerPinProperties := (Index := 72, Type_ := eControllerPinType.NA, Number := '175', Mapping := eControllerPinMappingType.CHA, Symbol := '175', Info := 'PIN_175', Description := 0);
  gc_Pin_C1_73 : TControllerPinProperties := (Index := 73, Type_ := eControllerPinType.DOU, Number := '149', Mapping := eControllerPinMappingType.FIX, Symbol := '149', Info := 'Blue fire', Description := 0);
  gc_Pin_C1_74 : TControllerPinProperties := (Index := 74, Type_ := eControllerPinType.DOU, Number := '173', Mapping := eControllerPinMappingType.FIX, Symbol := '173', Info := 'Orange flashing light', Description := 0);
  gc_Pin_C1_75 : TControllerPinProperties := (Index := 75, Type_ := eControllerPinType.DOU, Number := '152', Mapping := eControllerPinMappingType.FIX, Symbol := '152', Info := 'Supply Tor sensors', Description := 0);
  gc_Pin_C1_76 : TControllerPinProperties := (Index := 76, Type_ := eControllerPinType.DOU, Number := '176', Mapping := eControllerPinMappingType.FIX, Symbol := '176', Info := 'Overload security', Description := 0);
  gc_Pin_C1_77 : TControllerPinProperties := (Index := 77, Type_ := eControllerPinType.DOU, Number := '155', Mapping := eControllerPinMappingType.FIX, Symbol := '155', Info := 'Anti Startup', Description := 0);
  gc_Pin_C1_78 : TControllerPinProperties := (Index := 78, Type_ := eControllerPinType.DOU, Number := '179', Mapping := eControllerPinMappingType.FIX, Symbol := '179', Info := 'Ev Deviator Movements', Description := 0);
  gc_Pin_C1_79 : TControllerPinProperties := (Index := 79, Type_ := eControllerPinType.NA, Number := '158', Mapping := eControllerPinMappingType.CHA, Symbol := '158', Info := 'PIN_158', Description := 0);
  gc_Pin_C1_80 : TControllerPinProperties := (Index := 80, Type_ := eControllerPinType.DOU, Number := '182', Mapping := eControllerPinMappingType.FIX, Symbol := '182', Info := 'Ev Bypass', Description := 0);
  gc_Pin_C1_81 : TControllerPinProperties := (Index := 81, Type_ := eControllerPinType.DOU, Number := '251', Mapping := eControllerPinMappingType.FIX, Symbol := '251', Info := 'Ev Boost Regen cmd', Description := 0);
  gc_Pin_C1_82 : TControllerPinProperties := (Index := 82, Type_ := eControllerPinType.NA, Number := '238', Mapping := eControllerPinMappingType.CHA, Symbol := '238', Info := 'PIN_238', Description := 0);
  gc_Pin_C1_83 : TControllerPinProperties := (Index := 83, Type_ := eControllerPinType.DOU, Number := '252', Mapping := eControllerPinMappingType.FIX, Symbol := '252', Info := 'Return low side ev pro generator', Description := 0);
  gc_Pin_C1_84 : TControllerPinProperties := (Index := 84, Type_ := eControllerPinType.DOU, Number := '239', Mapping := eControllerPinMappingType.FIX, Symbol := '239', Info := 'PIN_239', Description := 0);
  gc_Pin_C1_85 : TControllerPinProperties := (Index := 85, Type_ := eControllerPinType.NA, Number := '253', Mapping := eControllerPinMappingType.CHA, Symbol := '253', Info := 'PIN_253', Description := 0);
  gc_Pin_C1_86 : TControllerPinProperties := (Index := 86, Type_ := eControllerPinType.NA, Number := '240', Mapping := eControllerPinMappingType.CHA, Symbol := '240', Info := 'PIN_240', Description := 0);
  gc_Pin_C1_87 : TControllerPinProperties := (Index := 87, Type_ := eControllerPinType.NA, Number := '254', Mapping := eControllerPinMappingType.CHA, Symbol := '254', Info := 'PIN_254', Description := 0);
  gc_Pin_C1_88 : TControllerPinProperties := (Index := 88, Type_ := eControllerPinType.NA, Number := '241', Mapping := eControllerPinMappingType.CHA, Symbol := '241', Info := 'PIN_241', Description := 0);
  gc_Pin_C1_89 : TControllerPinProperties := (Index := 89, Type_ := eControllerPinType.VOU, Number := '161', Mapping := eControllerPinMappingType.FIX, Symbol := '161', Info := 'Pvg Delta arm', Description := 0);
  gc_Pin_C1_90 : TControllerPinProperties := (Index := 90, Type_ := eControllerPinType.VOU, Number := '185', Mapping := eControllerPinMappingType.FIX, Symbol := '185', Info := 'Pvg arrow arm', Description := 0);
  gc_Pin_C1_91 : TControllerPinProperties := (Index := 91, Type_ := eControllerPinType.VOU, Number := '188', Mapping := eControllerPinMappingType.FIX, Symbol := '188', Info := 'Pvg telescope arm', Description := 0);
  gc_Pin_C1_92 : TControllerPinProperties := (Index := 92, Type_ := eControllerPinType.VOU, Number := '164', Mapping := eControllerPinMappingType.FIX, Symbol := '164', Info := 'Pvg prop Ev Tor', Description := 0);
  gc_Pin_C1_93 : TControllerPinProperties := (Index := 93, Type_ := eControllerPinType.DOU, Number := '191', Mapping := eControllerPinMappingType.FIX, Symbol := '191', Info := 'Suplly Pvg Delta Arm', Description := 0);
  gc_Pin_C1_94 : TControllerPinProperties := (Index := 94, Type_ := eControllerPinType.DOU, Number := '167', Mapping := eControllerPinMappingType.FIX, Symbol := '167', Info := 'Suplly Pvg Boom Arm', Description := 0);
  gc_Pin_C1_95 : TControllerPinProperties := (Index := 95, Type_ := eControllerPinType.DOU, Number := '194', Mapping := eControllerPinMappingType.FIX, Symbol := '194', Info := 'Suplly Pvg Telescope Arm', Description := 0);
  gc_Pin_C1_96 : TControllerPinProperties := (Index := 96, Type_ := eControllerPinType.DOU, Number := '170', Mapping := eControllerPinMappingType.FIX, Symbol := '170', Info := 'Suplly Pvg Prop Ev Tor', Description := 0);
END_VAR

FUNCTION MatchLibInit_Pins : BOOL

            gLib_MatchInitializer.PinConfigsPointer[0] := ADR(gc_ControllerPinConfigs);
gLib_MatchInitializer.PinConfigsInitializerCount := 1;
gLib_MatchInitializer.PinControllerCount[0] := 2;

          
END_FUNCTION
